// TIA Portal V16 export
// export: Created 2024-12-03T15:41:40.9629249Z, ExportSetting WithDefaults, DisplayName Totally Integrated Automation Portal, DisplayVersion V16 Update 6, DisplayName TIA Portal Version Control Interface, DisplayVersion V16 Update 2, DisplayName TIA Portal Openness, DisplayVersion V16 Update 6, DisplayName TIA Portal Teamcenter Gateway, DisplayVersion V16, DisplayName SINAMICS Startdrive Advanced, DisplayVersion V16 Update 5, DisplayName SINAMICS Startdrive G130, G150, S120, S150, SINAMICS MV, S210, DisplayVersion V16 Update 5, DisplayName SINAMICS Startdrive G110M, G120, G120C, G120D, G120P, G115D, DisplayVersion V16 Update 5, DisplayName STEP 7 Professional, DisplayVersion V16 Update 6, DisplayName STEP 7 Safety, DisplayVersion V16, DisplayName WinCC Advanced / Unified PC, DisplayVersion V16 Update 6
FUNCTION_BLOCK "SR"   // FB14, SCL
{ S7_Optimized_Access := 'FALSE' }
VERSION : 0.1
// stored: AutoNumber true, IsIECCheckEnabled false, SetENOAutomatically false, UDAEnableTagReadback false
   VAR_INPUT
      I_set : Bool;
      I_Reset : Bool;
   END_VAR
   VAR_OUTPUT
      O_StateExtend : "SmartBooldt";
      O_state : Bool;
   END_VAR
   VAR
      S_Reader { S7_SetPoint := 'True'} : "SmartBool";
   END_VAR
   VAR DB_SPECIFIC
      S_State : Bool;
   END_VAR
BEGIN
   IF #I_set THEN
       #S_State := true;
   END_IF;

   IF #I_Reset THEN
       #S_State := false;
   END_IF;

   #S_Reader(I_Sensor:= #S_State,O_data=> #O_StateExtend);

   #O_state := #O_StateExtend.State;
END_FUNCTION_BLOCK
